// TIA Portal project "2022.11.02—移动、转换" (V17)

(* hardware
DEVICE "S7-1200 station_1"  S7-1200 Station
   slot 0: "Rack_0"  S7-1200 Rack  Rack  V1.0
   slot 1: "PLC_1"  CPU 1214C DC/DC/Rly  6ES7 214-1HG40-0XB0  V4.5
*)

// ===== PLC "PLC_1"  CPU 1214C DC/DC/Rly =====

DATA_BLOCK "数据块_1"   // DB1
{ S7_Optimized_Access := 'TRUE' }
VERSION : 0.1
   VAR
      day_time : DTL;
      RETURN_VAL : Int;
      中间变量1 : DInt;
      中间变量2 : Real;
      中间变量3 : Real;
      中间变量4 : UDInt;
      中间变量5 : Real;
      中间变量6 : DInt;
      "Randow-score" : UDInt;
      待录入成绩 : UDInt;
      总成绩 : UDInt;
      平均值 : Real;
      取平均值 : Bool;
      随机生成成绩 : Bool;
      手动录入成绩 : Bool;
      操作数1 : Bool;
      操作数2 : Bool;
      操作数3 : Bool;
      运行标记 : UDInt;
      Score : Array[1..10] of UDInt;
      "index 1" : DInt := 1;
      "index 2" : DInt;
   END_VAR
BEGIN
END_DATA_BLOCK

ORGANIZATION_BLOCK "Main"   // OB1, LAD, ProgramCycle
TITLE = "Main Program Sweep (Cycle)"
{ S7_Optimized_Access := 'TRUE' }
VERSION : 0.1
   VAR_INPUT
      Initial_Call : Bool;   // Initial call of this OB
      Remanence : Bool;   // =True, if remanent data are available
   END_VAR
   VAR_TEMP   // added for the SCL form of the ladder/FBD networks
      _w1 : Bool;
      _w2 : Bool;
      _w3 : Bool;
      _w4 : Bool;
   END_VAR
BEGIN

REGION Network 1
   // 取纳秒前两个数或后两个数  用move取出 纳秒  conv转换类型      除数取前两位  取整
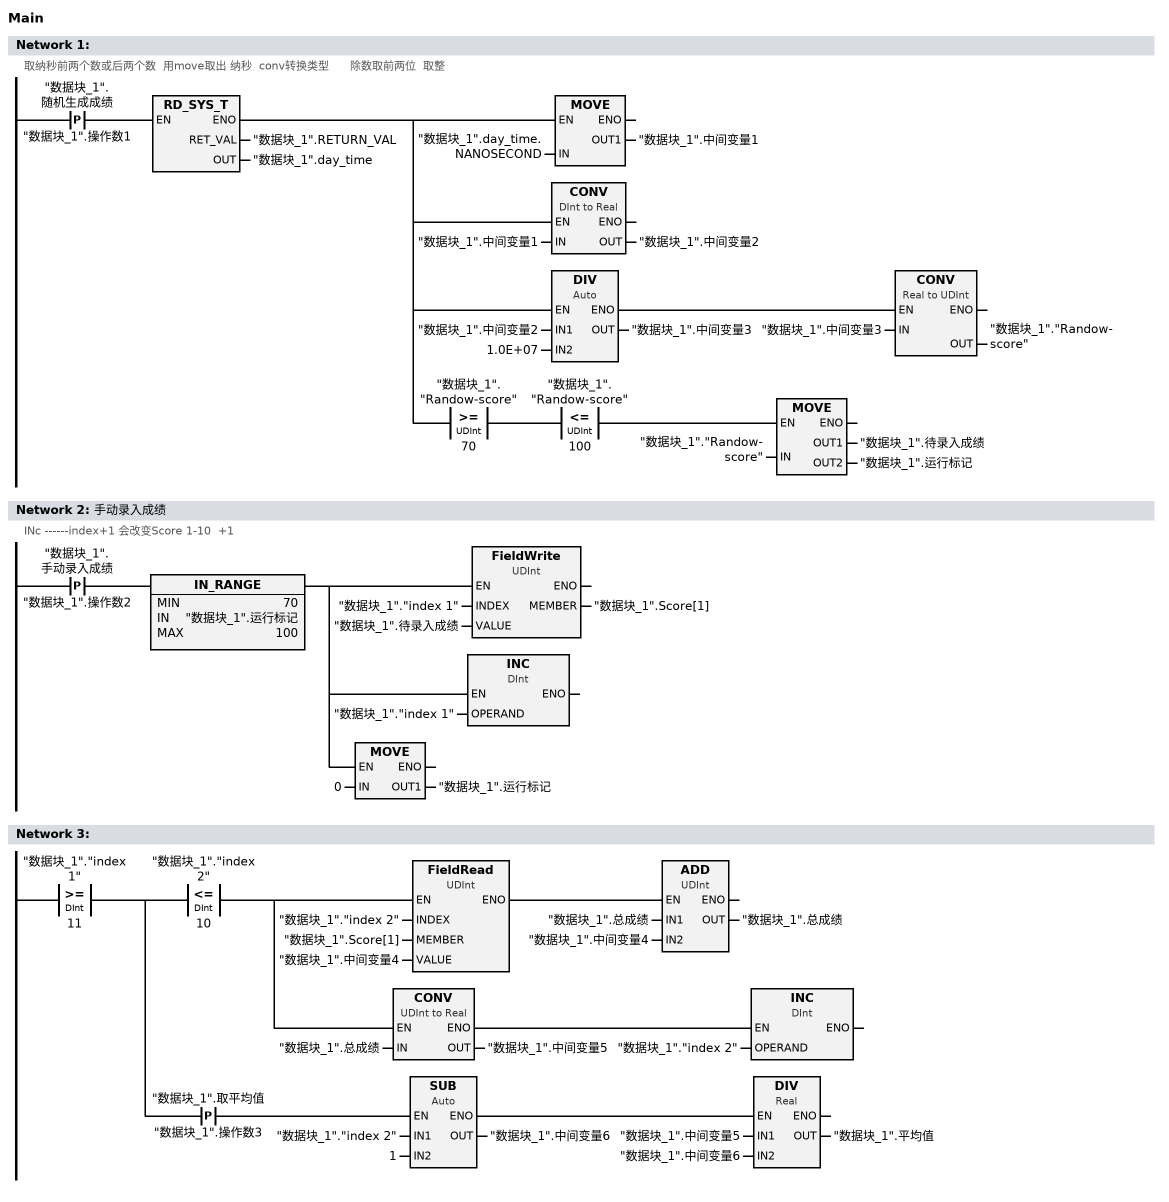
   // ENO of a box is taken as its EN; it also drops when the box reports an error
   #_w1 := "数据块_1".随机生成成绩 AND NOT "数据块_1".操作数1;   // rising edge of "数据块_1".随机生成成绩
   "数据块_1".操作数1 := "数据块_1".随机生成成绩;
   IF #_w1 THEN
       "数据块_1".RETURN_VAL := RD_SYS_T(OUT => "数据块_1".day_time);
       "数据块_1".中间变量1 := "数据块_1".day_time.NANOSECOND;
       "数据块_1".中间变量2 := DINT_TO_REAL("数据块_1".中间变量1);
       "数据块_1".中间变量3 := "数据块_1".中间变量2 / 1.0E+07;
       "数据块_1"."Randow-score" := REAL_TO_UDINT("数据块_1".中间变量3);
   END_IF;
   IF #_w1 AND ("数据块_1"."Randow-score" >= 70) AND ("数据块_1"."Randow-score" <= 100) THEN
       "数据块_1".待录入成绩 := "数据块_1"."Randow-score";
       "数据块_1".运行标记 := "数据块_1"."Randow-score";
   END_IF;
END_REGION

REGION Network 2: 手动录入成绩
   // INc ------index+1 会改变Score 1-10  +1
   // no SCL statement known for FieldWrite: written as a call
   #_w1 := "数据块_1".手动录入成绩 AND NOT "数据块_1".操作数2;   // rising edge of "数据块_1".手动录入成绩
   "数据块_1".操作数2 := "数据块_1".手动录入成绩;
   #_w2 := #_w1 AND (70 <= "数据块_1".运行标记) AND ("数据块_1".运行标记 <= 100);
   IF #_w2 THEN
       FieldWrite(index := "数据块_1"."index 1", value := "数据块_1".待录入成绩, member => "数据块_1".Score[1]);
       "数据块_1"."index 1" := "数据块_1"."index 1" + 1;
       "数据块_1".运行标记 := 0;
   END_IF;
END_REGION

REGION Network 3
   // no SCL statement known for FieldRead: written as a call
   // ENO of a box is taken as its EN; it also drops when the box reports an error
   #_w1 := "数据块_1"."index 1" >= 11;
   #_w2 := #_w1 AND ("数据块_1"."index 2" <= 10);
   #_w3 := #_w1 AND ("数据块_1"."index 2" <= 10);
   IF #_w3 THEN
       FieldRead(index := "数据块_1"."index 2", member := "数据块_1".Score[1], value := "数据块_1".中间变量4);
       "数据块_1".总成绩 := "数据块_1".总成绩 + "数据块_1".中间变量4;
   END_IF;
   IF #_w2 THEN
       "数据块_1".中间变量5 := UDINT_TO_REAL("数据块_1".总成绩);
       "数据块_1"."index 2" := "数据块_1"."index 2" + 1;
   END_IF;
   #_w4 := #_w1 AND "数据块_1".取平均值 AND NOT "数据块_1".操作数3;   // rising edge of "数据块_1".取平均值
   "数据块_1".操作数3 := "数据块_1".取平均值;
   IF #_w4 THEN
       "数据块_1".中间变量6 := "数据块_1"."index 2" - 1;
       "数据块_1".平均值 := "数据块_1".中间变量5 / "数据块_1".中间变量6;
   END_IF;
END_REGION
END_ORGANIZATION_BLOCK